# EPICS substitutions: tpmacApp/Db/pmacStatus.substitutions
file "db/pmacStatus.db"
{
pattern
{SYS,             PMAC,    VERSION  PLC  PORT,  NAXES }
{"XF:10IDA-CT",   "MC:2",  "1"      5    "P0",  8     }
}
